Universal Robots PolyScope program: test_script_calcs3.urp

Program test_script_calcs3 (installation=default directory=/programs createdIn=5.14.5 lastSavedIn=5.14.5 robotSerialNumber=20236801216)
Calibrated DH parameters: a=[-0.000021, -0.748897, -0.28186, -0.00004, -0.000055, 0]; d=[0.236225, -424.082933, -1564.66872, 1988.95162, 0.159094, 0.153873]; alpha=[1.570844, 0.001002, 0.000337, 1.571488, -1.569996, 0]; deltaTheta=[0, -0.516316, 5.626292, 1.173211, 0.000001, 0]
InitVariablesNode
Robot Program (runOnlyOnce=false)
  foo := 10
  Script: foo=42
  Script file /programs/pp11.script
    | pp11=p[1.1,0,0,0,0,0]
  Script file /programs/pp11ass.script
    | foo=pp11[0]
  Popup Message (haltProgram=false inputType=Variable) variable=foo
  Script file /programs/analyze_touchpoints.script
    | zcoord=p3[2]
    | l1p1x=p11[0]
    | l1p1y=p11[1]
